FUNCTION_BLOCK fbMainBlock
VAR_INPUT
END_VAR
VAR_OUTPUT
END_VAR
VAR_IN_OUT
	arstControl			: ARRAY[0..3] OF stControl;
	arstParams			: ARRAY[0..3] OF stParamschamber;
	arstInOuts			: ARRAY[0..3] OF stInOuts;
	stChamberTestParams : ARRAY[0..3] OF stTestParams;
END_VAR
VAR
	arFbChamber		: ARRAY[0..3] OF fbChamber;
	iSort			: INT;
	bTankBusy		: BOOL;
	bRealease40lTank	AT %Q* : BOOL;
END_VAR


//Bloki funkcyjne
arFbChamber[0](stControl:=arstControl[0],stInOuts:=arstInOuts[0],stParams:=arstParams[0],stChamberTestParams:=stChamberTestParams[arstParams[0].iCompresorType],stTime:=GVL_Aircom.stAC_DT_Data);
arFbChamber[1](stControl:=arstControl[1],stInOuts:=arstInOuts[1],stParams:=arstParams[1],stChamberTestParams:=stChamberTestParams[arstParams[1].iCompresorType],stTime:=GVL_Aircom.stAC_DT_Data);
arFbChamber[2](stControl:=arstControl[2],stInOuts:=arstInOuts[2],stParams:=arstParams[2],stChamberTestParams:=stChamberTestParams[arstParams[2].iCompresorType],stTime:=GVL_Aircom.stAC_DT_Data);
arFbChamber[3](stControl:=arstControl[3],stInOuts:=arstInOuts[3],stParams:=arstParams[3],stChamberTestParams:=stChamberTestParams[arstParams[3].iCompresorType],stTime:=GVL_Aircom.stAC_DT_Data);
//Obsługa kolejkowania
bTankBusy := arstControl[0].bTank40Used OR arstControl[1].bTank40Used OR arstControl[2].bTank40Used OR arstControl[3].bTank40Used;
IF NOT bTankBusy  THEN
	FOR iSort := 0 TO 3 DO
		IF arstControl[iSort].tActualTime<=arstControl[0].tActualTime AND arstControl[iSort].tActualTime<=arstControl[1].tActualTime AND arstControl[iSort].tActualTime<=arstControl[2].tActualTime AND arstControl[iSort].tActualTime<=arstControl[3].tActualTime AND arstControl[iSort].bStartPerform AND NOT arstControl[0].bStartAllow AND NOT arstControl[1].bStartAllow AND NOT arstControl[2].bStartAllow AND NOT arstControl[3].bStartAllow THEN
			arstControl[iSort].bStartAllow := TRUE;
		END_IF
		(*IF (arstControl[iSort].tActualTime<=arstControl[0].tActualTime AND arstControl[0].bStartPerform AND NOT arstControl[0].bStartAllow AND NOT arstControl[1].bStartAllow AND NOT arstControl[2].bStartAllow AND NOT arstControl[3].bStartAllow)
			AND (arstControl[iSort].tActualTime<=arstControl[1].tActualTime AND arstControl[1].bStartPerform AND NOT arstControl[0].bStartAllow AND NOT arstControl[1].bStartAllow AND NOT arstControl[2].bStartAllow AND NOT arstControl[3].bStartAllow) 
			AND (arstControl[iSort].tActualTime<=arstControl[2].tActualTime AND arstControl[2].bStartPerform AND NOT arstControl[0].bStartAllow AND NOT arstControl[1].bStartAllow AND NOT arstControl[2].bStartAllow AND NOT arstControl[3].bStartAllow) 
			AND (arstControl[iSort].tActualTime<=arstControl[3].tActualTime AND arstControl[3].bStartPerform AND NOT arstControl[0].bStartAllow AND NOT arstControl[1].bStartAllow AND NOT arstControl[2].bStartAllow AND NOT arstControl[3].bStartAllow) THEN
			arstControl[iSort].bStartAllow := TRUE;
		END_IF*)
	END_FOR
END_IF
bRealease40lTank := arstInOuts[0].bEjectPresure40 OR arstInOuts[1].bEjectPresure40 OR arstInOuts[2].bEjectPresure40 OR arstInOuts[3].bEjectPresure40;

END_FUNCTION_BLOCK

(* stored: Version 1.1.0.1, ProductVersion 3.1.4024.12
   POU fbMainBlock: Id {b41fe887-2897-4411-be45-b8590b9e5215}, SpecialFunc None *)
